Fanuc KAREL source: kt00017.KL

PROGRAM KT00017
%NOLOCKGROUP
VAR
Y1 : ARRAY[2] OF BYTE
I2:INTEGER
OUT:INTEGER
BEGIN
Y1[1]=2
I2=3
OUT=(Y1[1] + I2)
END KT00017
